TYPE "Fx_Types"
VERSION : 0.1
   STRUCT
      Enabled : Bool;
      Mode : Int;
      Setpoint : Real;   // generic setpoint
      Label : String[20];
   END_STRUCT;

END_TYPE
